TYPE ST_TwoHandOutCmd :
STRUCT
    StartAccepted : BOOL;
END_STRUCT
END_TYPE

(* stored: Version 1.1.0.1, ProductVersion 3.1.4024.12
   DUT ST_TwoHandOutCmd: Id {9cf1bd94-4ca5-47c5-876e-9843507105db} *)
